ABB RobotStudio station: assessment.rspag

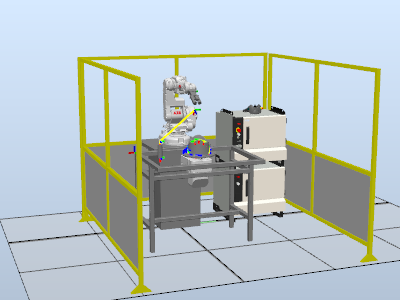
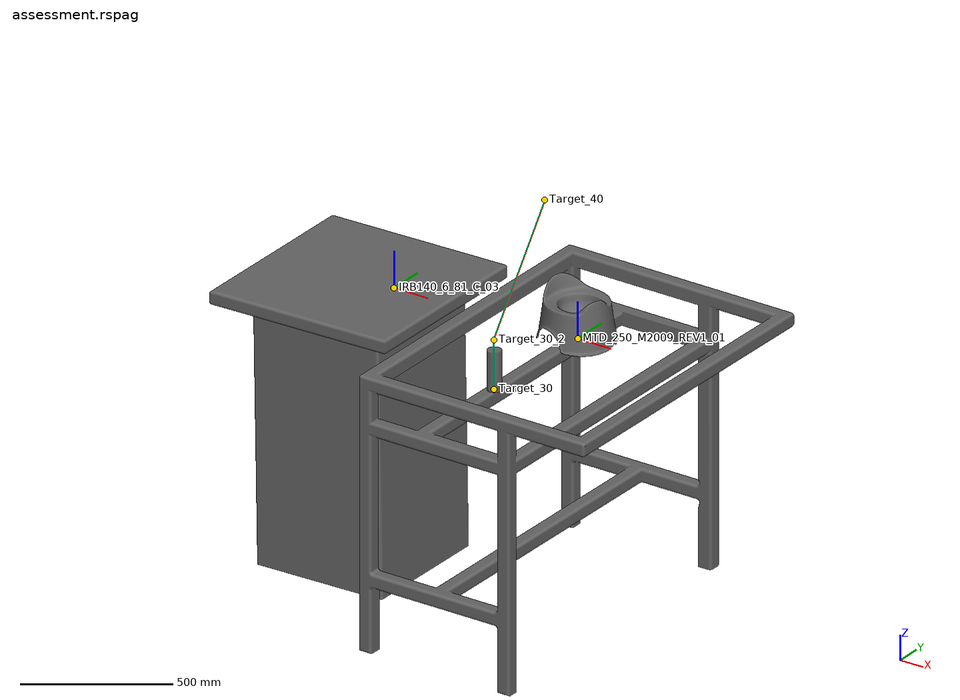
[picture v1: parts stored in the station drawn from their meshes, with robot base, taught points and paths (robot models come from the ABB library and are not in the file)]
--- station ---
Station ass-rs (saved by RobotStudio 22.3.10098.0)
Controller Controller, task T_ROB1: task frame (RAPID world) sits at (0, 0, 1000) mm in the station
Controller Controller
  mechanical unit ROB_1: IRB140_6_81_C_03, 6 joints, base frame (0, 0, 0) mm
  mechanical unit M7DM1: MTD_250_M2009_REV1_01, 1 joints, base frame (731.68, 0, 20) mm
Layout (positions relative to the parent item):
  - pedestal [part] at (-124.39, 0, -2.17) mm, rotated rx 0 ry -1 rz 0 deg, size 700 x 700 x 1000 mm
  - IRB140_6_81_C_03 [mechanism, from Robots\IRB140_6_81_C_G_03.rslib] at (0, 0, 1000) mm; joint values [0, 0, 0, 0, 0.5236, 0] (rad or m)
  - MTD_250_M2009_REV1_01 [mechanism] at (731.68, 0, 1020) mm; joint values [0] (rad or m)
      links: Base, Link1
  - table_2 [part] at (726.27, 0, 0) mm, size 900 x 1200 x 1000 mm
  - potty [part] at (844.34, 166.94, 1011.79) mm, rotated rx 90 ry 0 rz 0 deg, size 275.1 x 194.8 x 257.3 mm
  - holder [part] at (700, -430.42, 1000) mm, rotated rx 90 ry 0 rz 0 deg, size 50 x 120 x 49.5 mm
  - tool-m2 [part] at (700, -608.42, 1121) mm, size 50 x 50 x 143 mm
  - SmartComponent_1_2 [smart component, from Libraries\smart.rslib] at (506.29, 0, 1679.5) mm, rotated rx 180 ry 60 rz 180 deg
      connections:
        SmartComponent_1_2.opengrip -> Detacher.Execute
        SmartComponent_1_2.closegrip -> Attacher.Execute
    - smart [mechanism, from Libraries\smart.rslib] at (0, 0, 0) mm
    - Attacher [smart component, from Components\Attacher.rslib]
        properties: Parent=smart; Flange=0; Child=tool-m2; Mount=false; Offset=[0 0 0]; Orientation=[0 0 0]
    - Detacher [smart component, from Components\Detacher.rslib]
        properties: Child=tool-m2; KeepPosition=false
  - Fence_2500 [graphiccomponentgroup, from Equipment\Fence_2500.rslib] at (-700, -1000, 0) mm
    - Body 1 [part, from Equipment\Fence_2500.rslib]
    - Body 2 [part, from Equipment\Fence_2500.rslib]
  - Fence_2500_2 [graphiccomponentgroup, from Equipment\Fence_2500.rslib] at (-550, -1000, 0) mm, rotated rx 0 ry 0 rz -90 deg
    - Body 1 [part, from Equipment\Fence_2500.rslib]
    - Body 2 [part, from Equipment\Fence_2500.rslib]
  - IRC5_Dual-Cabinet [part, from Equipment\IRC5_Dual-Cabinet.rslib] at (0, 1000, 100) mm, rotated rx 90 ry 0 rz 90 deg
  - FlexPendant [part, from Equipment\FlexPendant.rslib] at (-144.27, 1016.87, 1340) mm, rotated rx -90 ry -15 rz 0 deg
  - Fence_2500_3 [graphiccomponentgroup, from Equipment\Fence_2500.rslib] at (-556.81, 1462.35, 0) mm, rotated rx 0 ry 0 rz -90 deg
    - Body 1 [part, from Equipment\Fence_2500.rslib]
    - Body 2 [part, from Equipment\Fence_2500.rslib]
Attachment: potty is attached to MTD_250_M2009_REV1_01 / Link1
Attachment: SmartComponent_1_2 is attached to IRB140_6_81_C_03 / Link6
Station logic (signal -> signal, property => property):
  Controller.opengripper -> SmartComponent_1_2.opengrip
  Controller.closegripper -> SmartComponent_1_2.closegrip

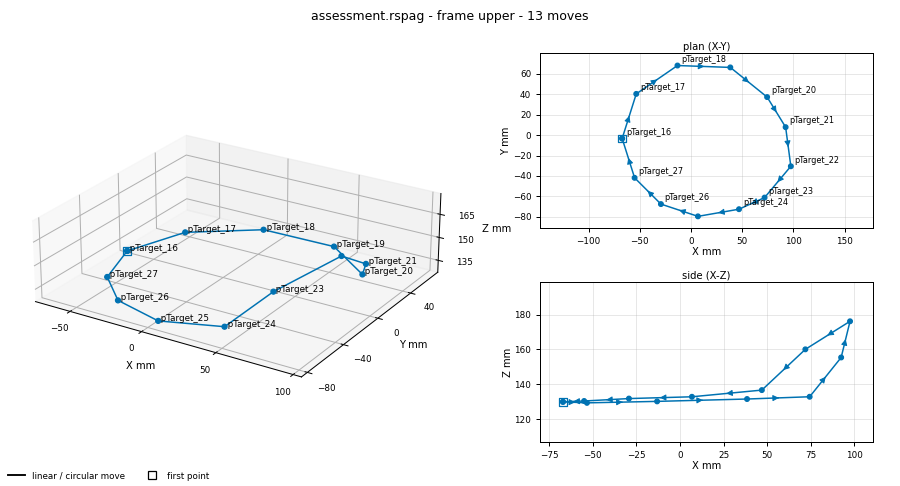
[picture p0: tool path of assessment.rspag in frame upper, 13 of 37 moves have a stored position in this frame; points joined in program order, loops and branches not executed]
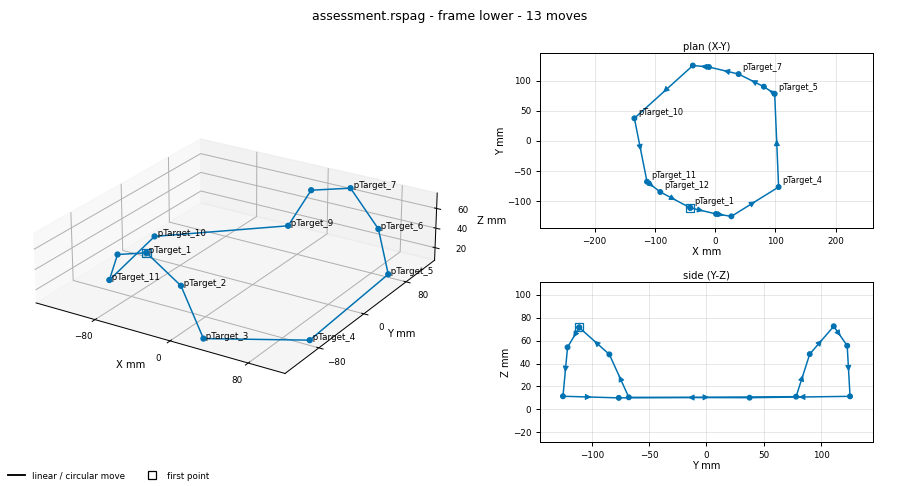
[picture p1: tool path of assessment.rspag in frame lower, 13 of 37 moves have a stored position in this frame; points joined in program order, loops and branches not executed]
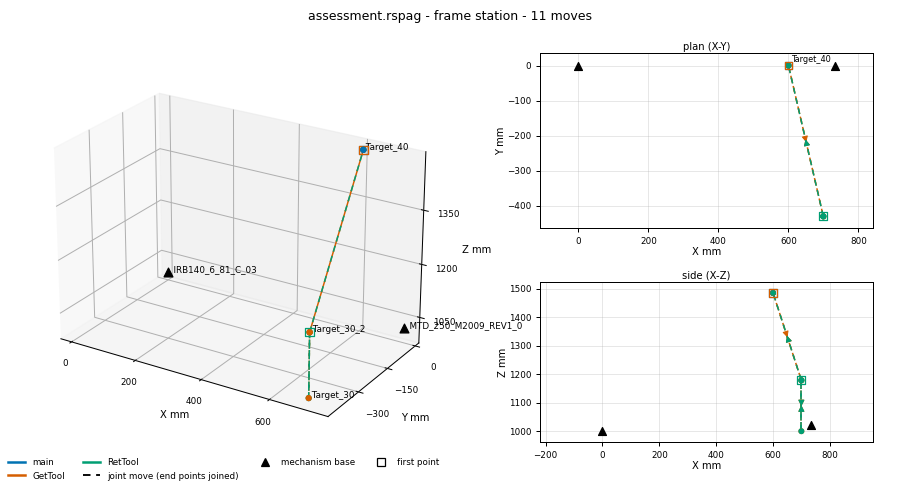
[picture p2: tool path of assessment.rspag in frame station, 11 of 37 moves have a stored position in this frame; points joined in program order, loops and branches not executed]
--- Backups/Controller/RAPID/TASK1/PROGMOD/CalibData.mod ---
MODULE CalibData
    PERS tooldata smart:=[TRUE,[[121,0,178],[1,0,0,0]],[1.5,[0,77,66],[1,0,0,0],0,0,0]];
    TASK PERS wobjdata upper:=[FALSE,FALSE,"M7DM1",[[-97.816751038,36.180264934,0],[0.372170585,0,0,-0.928164347]],[[0,0,0],[1,0,0,0]]];
    PERS tooldata gripped_pen:=[TRUE,[[121,0,178],[1,0,0,0]],[2,[0,50,88],[1,0,0,0],0,0,0]];
    TASK PERS wobjdata lower:=[FALSE,FALSE,"M7DM1",[[44.851962819,-51.238712166,0],[0.972480161,0,0,0.2329857]],[[0,0,0],[1,0,0,0]]];
    TASK PERS wobjdata holder:=[FALSE,TRUE,"ROB_1",[[326.436956592,-613.347606741,-0.000703581],[0.753365677,-0.00000134,-0.000003421,-0.657601822]],[[0,0,0],[1,0,0,0]]];
ENDMODULE

--- Backups/Controller/RAPID/TASK1/PROGMOD/Module1.mod ---
MODULE Module1
    CONST speeddata v480 := [480, 500, 5000, 1000];
    CONST speeddata v580 := [580, 500, 5000, 1000];
    CONST robtarget Target_10:=[[-43.065,-110.635,70.771],[0.209681593,0.707019727,0.577649194,-0.349968774],[0,0,0,0],[0,9E+09,9E+09,9E+09,9E+09,9E+09]];
    CONST robtarget Target_20:=[[3.692,-121.892,50.94],[0.100745288,0.558779008,0.682880562,-0.459663514],[0,0,0,0],[0,9E+09,9E+09,9E+09,9E+09,9E+09]];
    CONST robtarget Target_30:=[[-130.444414255,394.3057156,-0.573372141],[0.53270756,-0.46499376,0.532712398,0.464995655],[-1,-1,0,1],[0,9E+09,9E+09,9E+09,9E+09,9E+09]];
    CONST robtarget Target_40:=[[-570.763200944,353.875500921,485.714699934],[0.376679876,-0.569499214,0.652435525,0.328802071],[0,0,0,0],[0,9E+09,9E+09,9E+09,9E+09,9E+09]];
    CONST robtarget Target_50:=[[74.377,37.069,132.875],[0.160696902,0.872286571,0.135501229,-0.441511111],[0,0,0,0],[0,9E+09,9E+09,9E+09,9E+09,9E+09]];
    CONST robtarget Target_60:=[[92.447,7.687,155.419],[0.224143869,0.836516304,-0.286788219,-0.409576022],[0,0,0,0],[0,9E+09,9E+09,9E+09,9E+09,9E+09]];
    CONST robtarget Target_70:=[[97.541,-30.51,176.176],[0.073386891,-0.892538936,0.157378695,0.41619774],[0,0,0,0],[0,9E+09,9E+09,9E+09,9E+09,9E+09]];
    CONST robtarget Target_80:=[[71.907,-61.073,160.081],[0.272818606,-0.862822479,0.27619395,0.323765778],[0,0,0,0],[0,9E+09,9E+09,9E+09,9E+09,9E+09]];
    CONST robtarget Target_90:=[[46.937,-72.424,136.694],[0.304380715,-0.687064147,0.527202862,0.39667667],[0,0,0,0],[0,9E+09,9E+09,9E+09,9E+09,9E+09]];
    CONST robtarget Target_100:=[[6.819,-79.414,132.857],[0.383022221,-0.556670399,0.663413948,0.321393805],[0,0,0,0],[0,9E+09,9E+09,9E+09,9E+09,9E+09]];
    CONST robtarget Target_110:=[[-29.321,-67.434,131.833],[0.453153893,-0.365998151,0.784885567,0.211309131],[0,0,0,0],[0,9E+09,9E+09,9E+09,9E+09,9E+09]];
    CONST robtarget Target_120:=[[-55.033,-41.788,130.436],[0.483984059,-0.229273832,0.832847794,0.139848105],[0,0,0,0],[0,9E+09,9E+09,9E+09,9E+09,9E+09]];
    CONST robtarget Target_130:=[[-67.176,-3.375,129.955],[0.499524111,0.037775498,0.86520114,0.021809694],[0,0,0,0],[0,9E+09,9E+09,9E+09,9E+09,9E+09]];
    CONST robtarget pTarget_16:=[[-67.176,-3.375,129.955],[0.499524111,0.037775498,0.86520114,0.021809694],[-1,0,0,1],[0,9E+09,9E+09,9E+09,9E+09,9E+09]];
    CONST robtarget pTarget_17:=[[-53.413,40.181,129.372],[0.494668901,0.250398991,0.824563684,-0.112684317],[-1,0,-1,1],[27.69,9E+09,9E+09,9E+09,9E+09,9E+09]];
    CONST robtarget pTarget_18:=[[-13.158,67.869,130.217],[0.400997601,0.544003876,0.673133314,-0.30025364],[0,0,-1,1],[72.410892683,9E+09,9E+09,9E+09,9E+09,9E+09]];
    CONST robtarget pTarget_19:=[[38.446,66.026,131.57],[0.339011212,0.698627315,0.48388755,-0.40353948],[0,0,-1,1],[101.358206066,9E+09,9E+09,9E+09,9E+09,9E+09]];
    CONST robtarget pTarget_20:=[[74.377,37.069,132.875],[0.125560965,0.858966299,0.203522338,-0.452758213],[0,0,-1,1],[143.645323122,9E+09,9E+09,9E+09,9E+09,9E+09]];
    CONST robtarget pTarget_21:=[[92.447,7.687,155.419],[0.163510227,0.896108126,0.091118353,-0.402432699],[0,0,0,1],[150.907080035,9E+09,9E+09,9E+09,9E+09,9E+09]];
    CONST robtarget pTarget_22:=[[97.541,-30.51,176.176],[0.071353779,-0.865564483,0.200202369,0.453459783],[-1,0,0,1],[200.585872691,9E+09,9E+09,9E+09,9E+09,9E+09]];
    CONST robtarget pTarget_23:=[[71.907,-61.073,160.081],[0.263416226,-0.838230589,0.314810828,0.35899236],[0,0,-1,1],[239.048335885,9E+09,9E+09,9E+09,9E+09,9E+09]];
    CONST robtarget pTarget_24:=[[46.937,-72.424,136.694],[0.278478555,-0.740354901,0.450100432,0.414407911],[0,0,-1,1],[245.76126734,9E+09,9E+09,9E+09,9E+09,9E+09]];
    CONST robtarget pTarget_25:=[[6.819,-79.414,132.857],[0.356021117,-0.618157875,0.605300238,0.353187526],[-1,-1,0,1],[269.833066648,9E+09,9E+09,9E+09,9E+09,9E+09]];
    CONST robtarget pTarget_26:=[[-29.321,-67.434,131.833],[0.416411034,-0.463576336,0.728991937,0.283318879],[0,0,-1,1],[292.246516532,9E+09,9E+09,9E+09,9E+09,9E+09]];
    CONST robtarget pTarget_27:=[[-55.033,-41.788,130.436],[0.469129345,-0.326372089,0.797477351,0.193465221],[0,0,-1,1],[315.851943575,9E+09,9E+09,9E+09,9E+09,9E+09]];
    CONST robtarget pTarget_28:=[[-67.176,-3.375,129.955],[0.497545972,-0.103070716,0.856508879,0.090647526],[0,-1,0,1],[344.082220381,9E+09,9E+09,9E+09,9E+09,9E+09]];
    CONST robtarget pTarget_1:=[[-41.107,-110.971,71.542],[0.702561397,0.281958171,0.648459397,0.08004676],[-1,0,0,1],[-2.105914009,9E+09,9E+09,9E+09,9E+09,9E+09]];
    CONST robtarget pTarget_2:=[[1.584,-121.156,54.193],[0.675396677,0.156371296,0.689599897,0.209378434],[-1,-1,0,1],[-3.92180694,9E+09,9E+09,9E+09,9E+09,9E+09]];
    CONST robtarget pTarget_3:=[[27.028,-125.148,11.48],[0.653281482,0.092295955,0.701057385,0.27059805],[-1,0,0,1],[-32.551158425,9E+09,9E+09,9E+09,9E+09,9E+09]];
    CONST robtarget pTarget_4:=[[105.43,-76.46,10.079],[0.521333803,-0.15304592,0.690345527,0.477714418],[-1,-1,0,1],[-63.555127316,9E+09,9E+09,9E+09,9E+09,9E+09]];
    CONST robtarget pTarget_5:=[[98.908,78.149,11.135],[0.092295956,-0.560985527,0.430459333,0.701057385],[-1,-1,0,1],[-125.166946133,9E+09,9E+09,9E+09,9E+09,9E+09]];
    CONST robtarget pTarget_6:=[[80.955,90.057,48.248],[0.074256068,-0.571858441,0.415906147,0.703197011],[-1,-1,0,1],[-138.377102693,9E+09,9E+09,9E+09,9E+09,9E+09]];
    CONST robtarget pTarget_7:=[[39.047,111.017,72.521],[0.061628419,0.640856383,-0.298836237,-0.704416026],[-1,-1,0,1],[-142.703854651,9E+09,9E+09,9E+09,9E+09,9E+09]];
    CONST robtarget pTarget_8:=[[-10.219,122.737,55.527],[0.272570401,0.701333015,-0.090177616,-0.652461015],[-1,-1,0,1],[-200.125895099,9E+09,9E+09,9E+09,9E+09,9E+09]];
    CONST robtarget pTarget_9:=[[-36.921,125.206,11.41],[0.296103331,0.705209062,-0.059181007,-0.641483129],[-1,-1,0,1],[-178.997201013,9E+09,9E+09,9E+09,9E+09,9E+09]];
    CONST robtarget pTarget_10:=[[-133.959,37.599,10.238],[0.579227965,0.640856382,0.29883624,-0.405579787],[-1,-1,0,1],[-230.275801302,9E+09,9E+09,9E+09,9E+09,9E+09]];
    CONST robtarget pTarget_11:=[[-112.998,-67.723,10.56],[0.69636424,0.454519478,0.54167522,-0.122787804],[-1,-1,0,1],[-272.593504236,9E+09,9E+09,9E+09,9E+09,9E+09]];
    CONST robtarget pTarget_12:=[[-90.98,-84.69,47.986],[0.90360635,0.214264897,0.365950475,0.060550546],[-1,-1,0,1],[-298.481746114,9E+09,9E+09,9E+09,9E+09,9E+09]];
    CONST robtarget pTarget_13:=[[-41.293,-110.951,71.435],[0.704416026,0.298836239,0.640856382,0.061628417],[-1,-1,0,1],[-295.968321765,9E+09,9E+09,9E+09,9E+09,9E+09]];
    CONST robtarget Target_30_2:=[[-130.443175924,394.306159646,178.456398731],[0.53270756,-0.46499376,0.532712398,0.464995655],[-1,-1,0,1],[0,9E+09,9E+09,9E+09,9E+09,9E+09]];
!***********************************************************
    !
    ! Module:  Module1
    !
    ! Description:
    !   <Insert description here>
    !
    ! Author: sgmxu9
    !
    ! Version: 1.0
    !
    !***********************************************************


    !***********************************************************
    !
    ! Procedure main
    !
    !   This is the entry point of your program
    !
    !***********************************************************
    PROC main()
    !Add your code here
        ActUnit M7DM1;
        GetTool;
        UpperPath;
        MoveJ Target_40,v580,z100,smart\WObj:=holder;
        LowerPath;
        MoveJ Target_40,v580,z100,smart\WObj:=holder;
        RetTool;
    ENDPROC
    PROC UpperPath()
        MoveJ pTarget_16,v580,z100,smart\WObj:=upper;
        MoveL pTarget_17,v480,z100,smart\WObj:=upper;
        MoveL pTarget_18,v480,z100,smart\WObj:=upper;
        MoveL pTarget_19,v480,z100,smart\WObj:=upper;
        MoveL pTarget_20,v480,z100,smart\WObj:=upper;
        MoveL pTarget_21,v480,z100,smart\WObj:=upper;
        MoveL pTarget_22,v480,z100,smart\WObj:=upper;
        MoveL pTarget_23,v480,z100,smart\WObj:=upper;
        MoveL pTarget_24,v480,z100,smart\WObj:=upper;
        MoveL pTarget_25,v480,z100,smart\WObj:=upper;
        MoveL pTarget_26,v480,z100,smart\WObj:=upper;
        MoveL pTarget_27,v480,z100,smart\WObj:=upper;
        MoveL pTarget_28,v480,z100,smart\WObj:=upper;
    ENDPROC
    PROC LowerPath()
        MoveJ pTarget_1,v580,z100,smart\WObj:=lower;
        MoveL pTarget_2,v480,z100,smart\WObj:=lower;
        MoveL pTarget_3,v480,z100,smart\WObj:=lower;
        MoveL pTarget_4,v480,z100,smart\WObj:=lower;
        MoveL pTarget_5,v480,z100,smart\WObj:=lower;
        MoveL pTarget_6,v480,z100,smart\WObj:=lower;
        MoveL pTarget_7,v480,z100,smart\WObj:=lower;
        MoveL pTarget_8,v480,z100,smart\WObj:=lower;
        MoveL pTarget_9,v480,z100,smart\WObj:=lower;
        MoveL pTarget_10,v480,z100,smart\WObj:=lower;
        MoveL pTarget_11,v480,z100,smart\WObj:=lower;
        MoveL pTarget_12,v480,z100,smart\WObj:=lower;
        MoveL pTarget_13,v480,z100,smart\WObj:=lower;
    ENDPROC
    PROC GetTool()
        MoveJ Target_40,v580,z100,smart\WObj:=holder;
        MoveJ Target_30_2,v580,z100,smart\WObj:=holder;
        MoveJ Target_30,v580,z100,smart\WObj:=holder;
        WaitTime 1;
        CloseGrippers;
        MoveJ Target_30_2,v580,z100,smart\WObj:=holder;
        MoveJ Target_40,v580,z100,smart\WObj:=holder;
    ENDPROC
    PROC RetTool()
        MoveJ Target_30_2,v580,z100,smart\WObj:=holder;
        MoveJ Target_30,v580,z100,smart\WObj:=holder;
        WaitTime 1;
        OpenGrippers;
        MoveJ Target_30_2,v580,z100,smart\WObj:=holder;
        MoveJ Target_40,v580,z100,smart\WObj:=holder;
    ENDPROC
ENDMODULE

--- Backups/Controller/RAPID/TASK1/SYSMOD/gripper.sys ---
MODULE gripper(SYSMODULE,READONLY)
    PROC OpenGrippers()
        Reset closegripper;
        Set opengripper;
    ENDPROC
    PROC CloseGrippers()
        Reset opengripper;
        Set closegripper;
    ENDPROC
ENDMODULE

--- Backups/Controller/SYSPAR/EIO.cfg ---
EIO:CFG_1.0:6:1::
#
INDUSTRIAL_NETWORK:

      -Name "DeviceNet" -Label "DeviceNet Master/Slave Network" -Address "2"
#
DEVICENET_DEVICE:

      -Name "gripper_board" -VendorName "ABB Robotics"\
      -ProductName "24 VDC I/O Device" -Label "DSQC 652 24 VDC I/O Device"\
      -ProductCode 26 -DeviceType 7 -ConnectionType "COS" -OutputSize 2\
      -InputSize 2
#
DEVICENET_INTERNAL_DEVICE:

      -Name "DN_Internal_Device" -VendorName "ABB Robotics"\
      -ProductName "DeviceNet Internal Slave Device"
#
EIO_SIGNAL:

      -Name "opengripper" -SignalType "DO" -Device "gripper_board"\
      -DeviceMap "0" -Access "All"

      -Name "closegripper" -SignalType "DO" -Device "gripper_board"\
      -DeviceMap "1" -Access "All"
